(* Logix 5000 project; controller Lab1 vendor 1 type 14 code 155 rev 20.12; software revision 20.01 *)

TASK MainTask (continuous, watchdog 500 ms) : MainProgram

MODULES
   Local : vendor 1 type 14 code 155 (PointIO 0, rev 20.12)
      Kinetix_350 : vendor 1 type 37 code 27 (Ethernet 192.168.1.7, rev 1.1, MotionDiagnostics RPI 1 ms, MotionSync RPI 2 ms)
      XG_7702 : ETHERNET-MODULE (Ethernet 192.168.1.6, rev 1.1, Output RPI 10 ms)
      A_In : 1734-IE2V (PointIO 2, rev 3.1, Input RPI 80 ms)
      Stepper_1 : vendor 10 type 150 code 185 (PointIO 5, rev 1.1, Output RPI 50 ms)
      Stepper_2 : vendor 10 type 150 code 185 (PointIO 6, rev 1.1, Output RPI 50 ms)
      Discrete_IO : Embedded (PointIO 1, rev 20.11, Output RPI 20 ms)
      A_Out : 1734-OE2V (PointIO 3, rev 3.1, Output RPI 80 ms)
      HSC : vendor 1 type 109 code 13 (PointIO 4, rev 3.1, Output RPI 80 ms)
END_MODULES

VAR_GLOBAL   (* controller tags *)
   Axis : AXIS_CIP_DRIVE;
   Kinetix_350_Quick_Start : MOTION_GROUP;
END_VAR

PROGRAM MainProgram   (* main routine MainRoutine *)
VAR
   AXIS_MOTION_CONTROL : MOTION_INSTRUCTION;
   AXIS_MOTION_CONTROL_HOME : MOTION_INSTRUCTION;
   AXIS_MOTION_CONTROL_ON : MOTION_INSTRUCTION := (FLAGS := 301989888, ER := 1, ERR := 11);
   CAMERA_STATE : DINT;
   MASTER_DELAY : TIMER := (PRE := 500, ACC := 200);
   MASTER_STATE : DINT := 3;
   SORTED_DELAY : TIMER := (PRE := 500, ACC := 200);
   SORTED_POSITION : REAL := 1.0;
   SORTED_STATE : DINT;
   STEP_CONFIG_3401L : INT[8] := ([0] := -32592, [3] := 5); {constant}
   STEP_DISTANCE : DINT := 670;
   STEP_INCR_MOVE : INT[8] := ([0] := 2, [3] := 670, [4] := 2, [6] := 10, [7] := 10);
        [0]   // Incr Move
        [2]   // distance (x1000's) +
        [3]   // + distance (x1)
        [4]   // speed (x1000's) +
        [5]   // + speed (x1)
        [6]   // acc 10
        [7]   // dec 10
   STEP_MOVE : INT[8] := ([0] := 2, [3] := 670, [4] := 2, [6] := 10, [7] := 10);
        [0]   // Move type
        [2]   // 1000th place
        [3]   // 1s place pos
        [4]   // 1000th place
        [5]   // 1s place speed
        [6]   // Acc
        [7]   // Dec
   STEP_ONS1 : BOOL;
   STEP_ONS2 : BOOL;
   STEP_POSITION : DINT := 670;
   STEP_PRESET_3401L : INT[8] := ([0] := 512); {constant}
   STEP_PRESET_RESET_MOVE_COMPLETE : INT[8] := ([0] := 512);
   STEP_RESET_ERRORS_3401 : INT[8] := ([0] := 2048); {constant}
   STEP_SETPOINT : DINT;
   STEP_SPEED : DINT := 2000;
   STEP_STATE : DINT := 3;
   SYSTEM_COLOR : DINT;
   SYSTEM_DONE : BOOL;
   SYSTEM_NEXT : TIMER := (PRE := 200, ACC := 200, EN := 1, DN := 1);
END_VAR

ROUTINE CalculatePositionSpeed   (* structured text *)
   sbr();
   
   	STEP_POSITION := STEP_DISTANCE;
   
   	// Position
   	STEP_INCR_MOVE[2]:= STEP_POSITION / 1000;						// MSW integer divide
   	STEP_INCR_MOVE[3]:= STEP_POSITION - (STEP_INCR_MOVE[2] * 1000);	// LSW remainder
   
   	// Speed
   	STEP_INCR_MOVE[4]:= STEP_SPEED / 1000;							// MSW integer divide
   	STEP_INCR_MOVE[5]:= STEP_SPEED    - (STEP_INCR_MOVE[4] * 1000);	// LSW remainder
   
   ret();
END_ROUTINE

ROUTINE MainRoutine   (* ladder *)
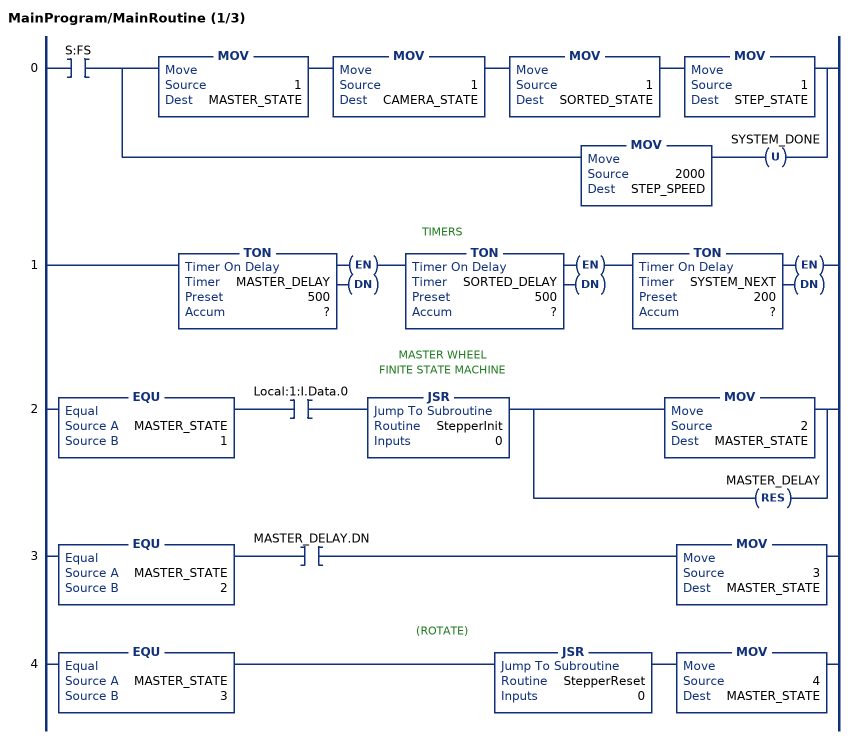
   0: XIC(S:FS)[MOV(1,MASTER_STATE) MOV(1,CAMERA_STATE) MOV(1,SORTED_STATE) MOV(1,STEP_STATE) ,MOV(2000,STEP_SPEED) OTU(SYSTEM_DONE) ];
   // TIMERS
   1: TON(MASTER_DELAY,?,?)TON(SORTED_DELAY,?,?)TON(SYSTEM_NEXT,?,?);
   // MASTER WHEEL
   // FINITE STATE MACHINE
   2: EQU(MASTER_STATE,1)XIC(Local:1:I.Data.0)JSR(StepperInit,0)[MOV(2,MASTER_STATE) ,RES(MASTER_DELAY) ];
   3: EQU(MASTER_STATE,2)XIC(MASTER_DELAY.DN)MOV(3,MASTER_STATE);
   // (ROTATE)
   4: EQU(MASTER_STATE,3)JSR(StepperReset,0)MOV(4,MASTER_STATE);
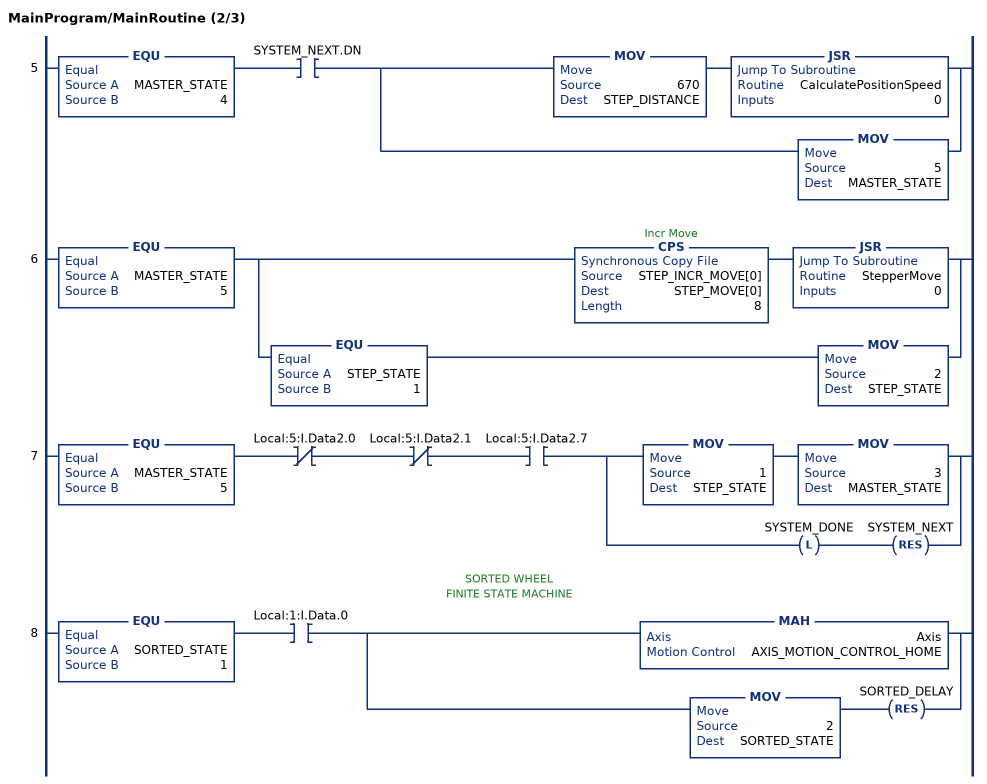
   5: EQU(MASTER_STATE,4)XIC(SYSTEM_NEXT.DN)[MOV(670,STEP_DISTANCE) JSR(CalculatePositionSpeed,0) ,MOV(5,MASTER_STATE) ];
   6: EQU(MASTER_STATE,5)[CPS(STEP_INCR_MOVE[0],STEP_MOVE[0],8) JSR(StepperMove,0) ,EQU(STEP_STATE,1) MOV(2,STEP_STATE) ];
   7: EQU(MASTER_STATE,5)XIO(Local:5:I.Data2.0)XIO(Local:5:I.Data2.1)XIC(Local:5:I.Data2.7)[MOV(1,STEP_STATE) MOV(3,MASTER_STATE) ,OTL(SYSTEM_DONE) RES(SYSTEM_NEXT) ];
   // SORTED WHEEL
   // FINITE STATE MACHINE
   8: EQU(SORTED_STATE,1)XIC(Local:1:I.Data.0)[MAH(Axis,AXIS_MOTION_CONTROL_HOME) ,MOV(2,SORTED_STATE) RES(SORTED_DELAY) ];
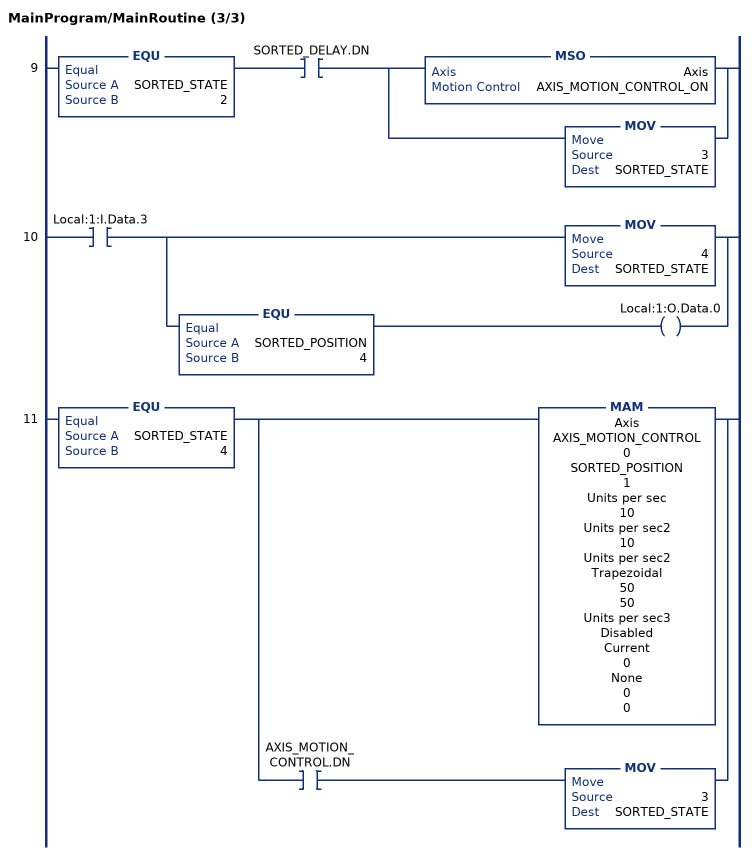
   9: EQU(SORTED_STATE,2)XIC(SORTED_DELAY.DN)[MSO(Axis,AXIS_MOTION_CONTROL_ON) ,MOV(3,SORTED_STATE) ];
   10: XIC(Local:1:I.Data.3)[MOV(4,SORTED_STATE) ,EQU(SORTED_POSITION,4) OTE(Local:1:O.Data.0) ];
   11: EQU(SORTED_STATE,4)[MAM(Axis,AXIS_MOTION_CONTROL,0,SORTED_POSITION,1,Units per sec,10,Units per sec2,10,Units per sec2,Trapezoidal,50,50,Units per sec3,Disabled,Current,0,None,0,0) ,XIC(AXIS_MOTION_CONTROL.DN) MOV(3,SORTED_STATE) ];
END_ROUTINE

ROUTINE StepperInit   (* ladder *)
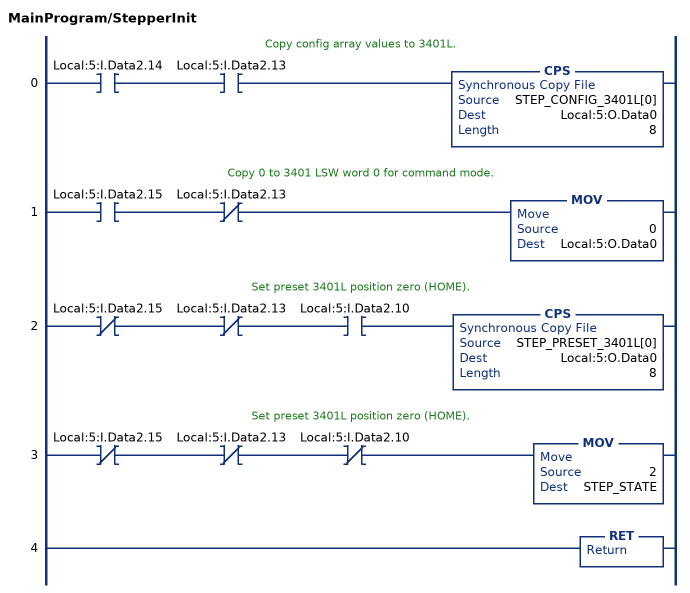
   // Copy config array values to 3401L.
   0: XIC(Local:5:I.Data2.14)XIC(Local:5:I.Data2.13)CPS(STEP_CONFIG_3401L[0],Local:5:O.Data0,8);
   // Copy 0 to 3401 LSW word 0 for command mode.
   1: XIC(Local:5:I.Data2.15)XIO(Local:5:I.Data2.13)MOV(0,Local:5:O.Data0);
   // Set preset 3401L position zero (HOME).
   2: XIO(Local:5:I.Data2.15)XIO(Local:5:I.Data2.13)XIC(Local:5:I.Data2.10)CPS(STEP_PRESET_3401L[0],Local:5:O.Data0,8);
   // Set preset 3401L position zero (HOME).
   3: XIO(Local:5:I.Data2.15)XIO(Local:5:I.Data2.13)XIO(Local:5:I.Data2.10)MOV(2,STEP_STATE);
   4: RET();
END_ROUTINE

ROUTINE StepperMove   (* ladder *)
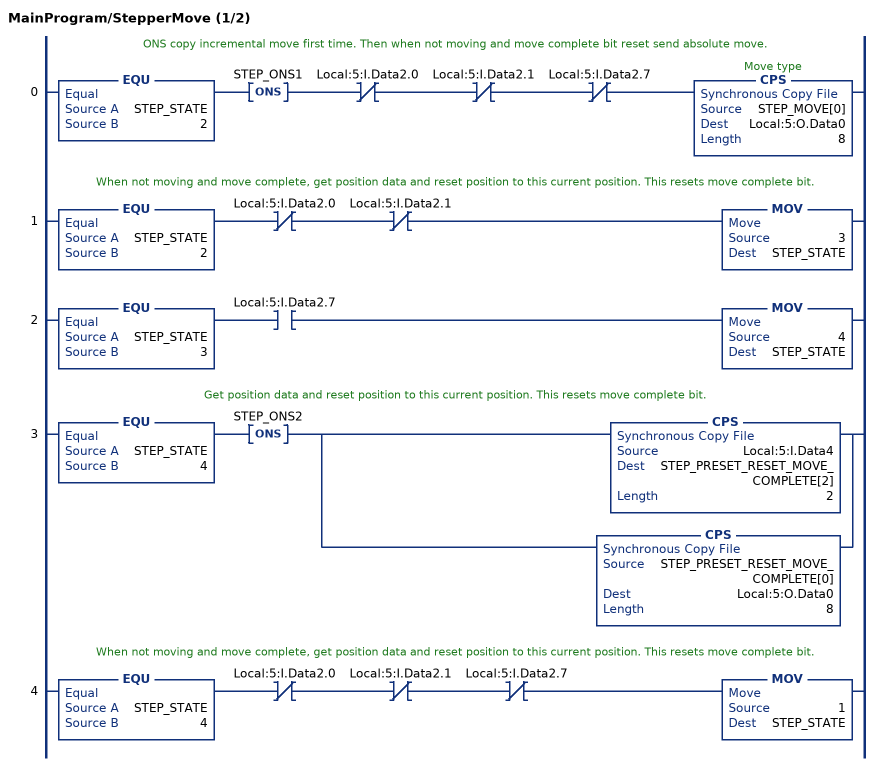
   // ONS copy incremental move first time. Then when not moving and move complete bit reset send absolute move.
   0: EQU(STEP_STATE,2)ONS(STEP_ONS1)XIO(Local:5:I.Data2.0)XIO(Local:5:I.Data2.1)XIO(Local:5:I.Data2.7)CPS(STEP_MOVE[0],Local:5:O.Data0,8);
   // When not moving and move complete, get position data and reset position to this current position. This resets move complete bit.
   1: EQU(STEP_STATE,2)XIO(Local:5:I.Data2.0)XIO(Local:5:I.Data2.1)MOV(3,STEP_STATE);
   2: EQU(STEP_STATE,3)XIC(Local:5:I.Data2.7)MOV(4,STEP_STATE);
   // Get position data and reset position to this current position. This resets move complete bit.
   3: EQU(STEP_STATE,4)ONS(STEP_ONS2)[CPS(Local:5:I.Data4,STEP_PRESET_RESET_MOVE_COMPLETE[2],2) ,CPS(STEP_PRESET_RESET_MOVE_COMPLETE[0],Local:5:O.Data0,8) ];
   // When not moving and move complete, get position data and reset position to this current position. This resets move complete bit.
   4: EQU(STEP_STATE,4)XIO(Local:5:I.Data2.0)XIO(Local:5:I.Data2.1)XIO(Local:5:I.Data2.7)MOV(1,STEP_STATE);
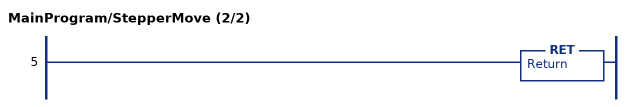
   5: RET();
END_ROUTINE

ROUTINE StepperReset   (* ladder *)
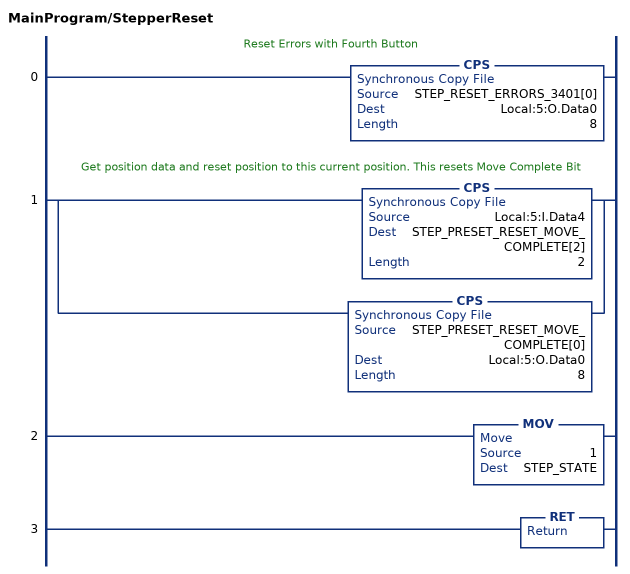
   // Reset Errors with Fourth Button
   0: CPS(STEP_RESET_ERRORS_3401[0],Local:5:O.Data0,8);
   // Get position data and reset position to this current position. This resets Move Complete Bit
   1: [CPS(Local:5:I.Data4,STEP_PRESET_RESET_MOVE_COMPLETE[2],2) ,CPS(STEP_PRESET_RESET_MOVE_COMPLETE[0],Local:5:O.Data0,8) ];
   2: MOV(1,STEP_STATE);
   3: RET();
END_ROUTINE
END_PROGRAM
